// TIA Portal V19 export
FUNCTION_BLOCK "ButtonsSafe_LB212_FeedA02"   // FB161, LAD
TITLE = LB212 SAFE BUTTONS (@ Flying Cut) used for feed Area 02 material
// stored: MemoryReserve 100, SetENOAutomatically false
   VAR_INPUT
      Reset_OthersPBs_Activation_IN : Bool := FALSE;
   END_VAR
   VAR_OUTPUT
      Reset_OthersPBs_Activation_OUT : Bool;
   END_VAR
   VAR
      i : Int;
      iOperation : Int;
      iConcurrentOperation : Int;
      SettingWriteDone : Bool;
      PbPanel : "Buttons2Hands";
      PB : Struct
         ResetAlarms : Bool;
         Rollformer_Bwd : Bool;
         Rollformer_Fwd : Bool;
      END_STRUCT;
   END_VAR
   VAR CONSTANT
      ITEMS : Int := 2;
      ROLLFORMER_BWD : Int := 1;
      ROLLFORMER_FWD : Int := 2;
   END_VAR
BEGIN

REGION Network 1 (SCL): Interlocks between operations selected
   IF "Area02".AreaInterface.ManOneShot THEN
       #SettingWriteDone := FALSE;
   END_IF;

   // Interblocco tra operazioni
   // 
   IF NOT #SettingWriteDone THEN
       #SettingWriteDone := TRUE;

       FOR #iOperation := 1 TO #ITEMS DO
           FOR #iConcurrentOperation := 1 TO #ITEMS DO
               #PbPanel.Enables[#iOperation, #iConcurrentOperation] := FALSE;
           END_FOR;
       END_FOR;

   END_IF;
END_REGION

REGION Network 2 (SCL): Buttons for Op selection
   #PbPanel.Buttons[ROLLFORMER_BWD] := "LB212_RollFormer_Pb_BWD";
   #PbPanel.Buttons[ROLLFORMER_FWD] := "LB212_RollFormer_Pb_FWD";
END_REGION

REGION Network 3 (SCL): Operation enable
   #PbPanel.OpEnabled[ROLLFORMER_BWD] := "Rollformer".COut.Feed.Bwd_CheckNext;
   #PbPanel.OpEnabled[ROLLFORMER_FWD] := "Rollformer".COut.Feed.Fwd_CheckNext;
END_REGION

REGION Network 4 (SCL): Operation running
   #PbPanel.OpRunning[ROLLFORMER_BWD] := "Rollformer".COut.Feed.VelBwd_Running;
   #PbPanel.OpRunning[ROLLFORMER_FWD] := "Rollformer".COut.Feed.VelFwd_Running OR "Rollformer".COut.Feed.PosFwd_Running;
END_REGION

REGION Network 5 (SCL): Operation done
   #PbPanel.OpDone[ROLLFORMER_BWD] := FALSE;
   #PbPanel.OpDone[ROLLFORMER_FWD] := "Rollformer".COut.Feed.InPosition;
END_REGION

REGION Network 6: Main
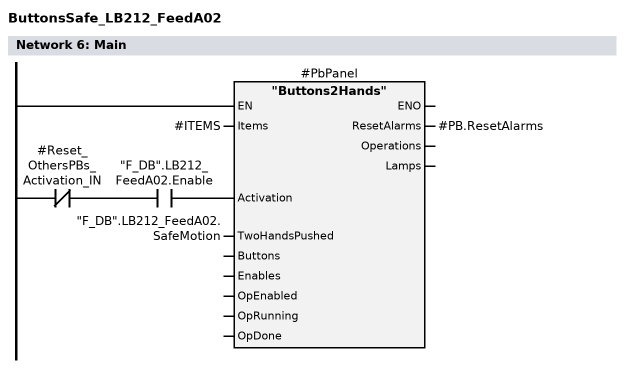
   RUNG wire#powerrail
      #PbPanel(Activation := wire#w1, Items := #ITEMS, TwoHandsPushed := "F_DB".LB212_FeedA02.SafeMotion, Buttons :=, Enables :=, OpEnabled :=, OpRunning :=, OpDone :=, ResetAlarms => #PB.ResetAlarms, Operations =>, Lamps =>)
   END_RUNG
   RUNG wire#powerrail
      I_Contact( #Reset_OthersPBs_Activation_IN )
      Contact( "F_DB".LB212_FeedA02.Enable )
   END_RUNG wire#w1
   // the same network as SCL:
   #PbPanel(Items := #ITEMS,   // "Buttons2Hands"
            Activation := NOT #Reset_OthersPBs_Activation_IN AND "F_DB".LB212_FeedA02.Enable,
            TwoHandsPushed := "F_DB".LB212_FeedA02.SafeMotion,
            ResetAlarms => #PB.ResetAlarms);
END_REGION

REGION Network 7 (SCL): Safe Buttons
   #PB.Rollformer_Bwd := #PbPanel.Operations[ROLLFORMER_BWD];
   #PB.Rollformer_Fwd := #PbPanel.Operations[ROLLFORMER_FWD];
END_REGION

REGION Network 8 (SCL): Lamp selection
   "LB212_RollFormer_Lp_BWD" := #PbPanel.Lamps[ROLLFORMER_BWD];
   "LB212_RollFormer_Lp_FWD" := #PbPanel.Lamps[ROLLFORMER_FWD];
END_REGION

REGION Network 9 (SCL): Reset others safe push buttons activation / execution
   #Reset_OthersPBs_Activation_OUT := FALSE;

   FOR #i := 1 TO #ITEMS DO

       IF #PbPanel.Buttons[#i] OR #PbPanel.Operations[#i] THEN
           #Reset_OthersPBs_Activation_OUT := TRUE;
           EXIT;
       END_IF;

   END_FOR;
END_REGION

REGION Network 10: >
END_REGION

REGION Network 11: >
END_REGION

REGION Network 12: >
END_REGION
END_FUNCTION_BLOCK
